FUNCTION F_Concat3 : T_MaxString
VAR_INPUT
	StringOne 	: STRING;
	StringTwo	: STRING;
	StringThree	: STRING;
END_VAR
VAR
	response : T_MaxString;
END_VAR

response := concat(StringOne, StringTwo);
response := concat(response, StringThree);
F_Concat3 := response;

END_FUNCTION

(* stored: Version 1.1.0.1, ProductVersion 3.1.4020.12
   POU F_Concat3: Id {88f226d8-71b0-47f7-94e2-4553db7f68e1}, SpecialFunc None *)
